Staubli VAL3: calculate_total.pgx

program calculate_total(num x_nNum_choose, num& x_nNum_total)
  local num l_nNum_lCol
  local num l_nNum_lRow
begin
  call return_config(x_nNum_choose,l_nNum_lRow,l_nNum_lCol)
    //(max index)
  x_nNum_total = (l_nNum_lRow + 1) * (l_nNum_lCol+1)
end
